(* Logix 5000 project; controller WWTP_SOLIDS_CLX vendor 1 type 14 code 54 rev 17.2; software revision 17.00; part 4 of 16 *)

ADD_ON_INSTRUCTION P_DoseFM   (* revision 0.12, ExecutePrescan, ExecuteEnableInFalse *)
// Dosing with Flowmeter
// Revision note:
// Cleaned up rate, qty code; added checks for Inp PVs being Infinite or Not A Number.
// Help:
// This Instruction monitors a flowmeter which provides flow rate (AI),
// quantity pulses (e.g., 1756-CFM/HSC), or rate and total (fieldbus),
// and provides:
// *  Optional integration (totalizing) of analog flow to a Quantity
// *  Optional differentiation of pulse count or quantity to a flow Rate
// *  Commands to Start, Stop and Clear the Quantity (total)
// *  Outputs to run and clear an external totalizer (e.g. on a fieldbus flowmeter)
// *  Commands to Start and Stop Flow for a dose
// *  Optional switching to a slow delivery (dribble) when approaching setpoint
// *  Stopping flow just before reaching setpoint using a Preact value
// *  Optional automatic adjustment of the preact value to fine tune the stop point
// *  Commands to check if the delivered quantity is within user-specified tolerances and alarm if not
// *  Program and Operator Settings for Setpoint, Preact, Dribble Quantity, High and Low Tolerances
// *  Zero failure alarm if quantity does not zero when totalizer is cleared
// *  Configurable Low Flow Cutoff to account for zero error on analog flowmeters
// *  Conversion of flow units to alternate quantity units (say, GPM to Barrels)
// *  Monitoring of input communication status
// *  Mode selection (Operator, Program or Maintenance)
// *  Simulation using configured simulated Delivery Rate and simulated Dribble Rate
VAR_INPUT
   Inp_RatePV : REAL; {visible}   // Flow Rate from Flowmeter (EU/time, see Cfg_RateTime)
   Inp_QtyPV : REAL; {visible}   // Quantity from Flowmeter (EU or Pulse Count)
   Inp_RatePVBad : BOOL;   // 1=Rate PV Input Quality = Bad (fail)
   Inp_RatePVUncertain : BOOL;   // 1=Rate PV Input Quality = Uncertain
   Inp_QtyPVBad : BOOL;   // 1=Quantity PV Input Quality = Bad (fail)
   Inp_QtyPVUncertain : BOOL;   // 1=Quantity PV Input Quality = Uncertain
   Inp_CtrldEqpFault : BOOL; {visible}   // Controlled Equipment device or I/O status 0=OK, 1=fail
   Inp_Sim : BOOL;   // 1=Simulate working flowmeter; 0=use actual flowmeter
   Inp_Reset : BOOL; {visible}   // 1=Reset all fault conditions and latched Alarms
   Cfg_HasDribble : BOOL;   // 1=Slow to Dribble before complete, 0=use complete only
   Cfg_AutoAdjPreact : BOOL;   // 1=enable automatic adjustment of preact after each delivery
   Cfg_CalcRate : BOOL := 1;   // 1=differentiate Inp_Qty to get rate, 0=use Inp_Rate
   Cfg_CalcQty : BOOL;   // 1=integrate Inp_Rate to get Quantity, 0=use Inp_Qty
   Cfg_SetTrack : BOOL := 1;   // 1=PSets track OSets in Oper, OSets track PSets in Prog, 0=no tracking
   Cfg_PCmdClear : BOOL := 1;   // 1=Clear Program Commands on receipt 0=Leave Set
   Cfg_HasOverTolAlm : BOOL;   // 1=Over Tolerance Alarm exists and will be checked
   Cfg_HasUnderTolAlm : BOOL;   // 1=Under Tolerance Alarm exists and will be checked
   Cfg_HasZeroFaultAlm : BOOL;   // 1=Zero Fault Alarm exists and will be checked
   Cfg_HasEqpFaultAlm : BOOL;   // 1=Equipment Fault Alarm exists and will be checked
   Cfg_OverTolResetReqd : BOOL;   // 1=Reset requied to clear Out of Tolerance High Alarm
   Cfg_UnderTolResetReqd : BOOL;   // 1=Reset required to clear Out of Tolerance Low Alarm
   Cfg_ZeroFaultResetReqd : BOOL;   // 1=Reset required to clear Zero Fault Alarm
   Cfg_EqpFaultResetReqd : BOOL;   // 1=Reset required to clear Equipment Fault Alarm
   Cfg_OverTolAckReqd : BOOL := 1;   // 1=Acknowledge required for Out of Tolerance High Alarm
   Cfg_UnderTolAckReqd : BOOL := 1;   // 1=Acknowledge required for Out of Tolerance Low Alarm
   Cfg_ZeroFaultAckReqd : BOOL := 1;   // 1=Acknowledge required for Zero Fault Alarm
   Cfg_EqpFaultAckReqd : BOOL := 1;   // 1=Acknowledge required for Equipment Fault Alarm
   Cfg_OverTolSeverity : SINT := 3;   // Over Tolerance Alarm Severity 1=info, 2=warn, 3=excep, 4=fault
   Cfg_UnderTolSeverity : SINT := 2;   // Under Tolerance Alarm Severity 1=info, 2=warn, 3=excep, 4=fault
   Cfg_ZeroFaultSeverity : SINT := 4;   // Zero Fault Alarm Severity 1=info, 2=warn, 3=excep, 4=fault
   Cfg_EqpFaultSeverity : SINT := 4;   // Equipment Fault Alarm Severity 1=info, 2=warn, 3=excep, 4=fault
   Cfg_MaxQty : REAL := 1.5e+38;   // Maximum allowed quantity to deliver (setpoint) (EU)
   Cfg_EUQtyMult : REAL := 1.0;   // Rate to Quantity EU Multiplier (e.g., Gal to Bbl.)
   Cfg_Rollover : REAL;   // Quantity Rollover (e.g., total counts for pulse input)
   Cfg_CountsPerEU : REAL := 1.0;   // Number of Counts in Inp_QtyPV which equal 1.0 EU
   Cfg_RateTime : REAL := 1.0;   // Time factor for rate (60 for /min, 3600 for /hr) (Sec)
   Cfg_RateFiltTC : REAL := 0.1;   // Filter Time Constant (sec) for calculated Rate
   Cfg_LoRateCutoff : REAL;   // Rate below which to report zero flow (Inp_RatePV untis)
   Cfg_BumpT : REAL;   // Bump (manual top-off) Time (Sec)
   Cfg_AutoAdjPct : REAL := 10.0;   // Percentage of delivery error to auto-adjust preact (%)
   Cfg_SimRate : REAL := 1.0;   // Rate at which to deliver when running in Simulation (EU/rate time)
   Cfg_SimDribbleRate : REAL := 0.1;   // Rate at which to dribble when running in Simulation (EU/rate time)
   Cfg_ClearPulseT : DINT := 1;   // Time to pulse Out_Clear to clear external totalizer (sec)
   PSet_SP : REAL;   // Program Setting of total quantity to deliver (EU)
   PSet_DribbleQty : REAL;   // Program Setting of quantity to dribble (EU)
   PSet_Preact : REAL;   // Program Setting of amount before total to stop flow (EU)
   PSet_TolHi : REAL;   // Program Setting of High Tolerance Limit (OK amount > SP)
   PSet_TolLo : REAL;   // Program Setting of Low Tolerance Limit (OK amount < SP)
   PSet_Owner : DINT;   // Program Owner Request ID (non-zero) or Release (zero)
   OSet_SP : REAL;   // Operator Setting of total quantity to deliver (EU)
   OSet_DribbleQty : REAL;   // Operator Setting of quantity to dribble (EU)
   OSet_Preact : REAL;   // Operator Setting of amount before total to stop flow (EU)
   OSet_TolHi : REAL;   // Operator Setting of High Tolerance Limit (OK amount > SP)
   OSet_TolLo : REAL;   // Operator Setting of Low Tolerance Limit (OK amount < SP)
   PCmd_ClearTot : BOOL;   // Program Command to Clear Totalizer Qty
   PCmd_StartTot : BOOL;   // Program Command to Start Totalizer
   PCmd_StopTot : BOOL;   // Program Command to Stop Totalizer
   PCmd_StartFlow : BOOL;   // Program Command to Start Delivery
   PCmd_StopFlow : BOOL;   // Program Command to Stop/Pause Delivery
   PCmd_CheckTol : BOOL;   // Program Command to Check Tolerances
   PCmd_Acq : BOOL;   // Program Command to Acquire ownership (Oper/OOS to Prog)
   PCmd_Rel : BOOL;   // Program Command to Release ownership (Prog to OOS)
   PCmd_Lock : BOOL;   // Program Command to Lock Mode in Prog
   PCmd_Unlock : BOOL;   // Program Command to Unlock Mode
   PCmd_Reset : BOOL;   // Program Command to Reset all Alarms requiring Reset
   PCmd_OverTolAck : BOOL;   // Program Command to Acknowledge Out of Tolerance High Alarm
   PCmd_OverTolInhibit : BOOL;   // Program Command to Inhibit Out of Tolerance High Alarm
   PCmd_OverTolUninhibit : BOOL;   // Program Command to Uninhibit Out of Tolerance High Alarm
   PCmd_UnderTolAck : BOOL;   // Program Command to Acknowledge Out of Tolerance Low Alarm
   PCmd_UnderTolInhibit : BOOL;   // Program Command to Inhibit Out of Tolerance Low Alarm
   PCmd_UnderTolUninhibit : BOOL;   // Program Command to Uninhibit Out of Tolerance Low Alarm
   PCmd_ZeroFaultAck : BOOL;   // Program Command to Acknowledge Zero Fault Alarm
   PCmd_ZeroFaultInhibit : BOOL;   // Program Command to Inhibit Zero Fault Alarm
   PCmd_ZeroFaultUninhibit : BOOL;   // Program Command to Uninhibit Zero Fault Alarm
   PCmd_EqpFaultAck : BOOL;   // Program Command to Acknowledge Equipment Fault Alarm
   PCmd_EqpFaultInhibit : BOOL;   // Program Command to Inhibit Equipment Fault Alarm
   PCmd_EqpFaultUninhibit : BOOL;   // Program Command to Uninhibit Equipment Fault Alarm
   OCmd_ClearTot : BOOL;   // Operator Command to Clear Totalizer Qty
   OCmd_StartTot : BOOL;   // Operator Command to Start Totalizer
   OCmd_StopTot : BOOL;   // Operator Command to Stop Totalizer
   OCmd_StartFlow : BOOL;   // Operator command to Start Deliver
   OCmd_StopFlow : BOOL;   // Operator Command to Stop/Pause Delivery
   OCmd_CheckTol : BOOL;   // Operator Command to Check Tolerances
   OCmd_Bump : BOOL;   // Operator Command to Bump Delivery for Under Tolerance
   OCmd_Reset : BOOL;   // Operator Command to Reset all Alarms requiring Reset
END_VAR
VAR_OUTPUT
   Out_RunFlow : BOOL; {visible}   // 1=Deliver at Full (fast) Flow
   Out_DribbleFlow : BOOL; {visible}   // 1=Deliver at Dribble (slow) Flow
   Out_StopFlow : BOOL; {visible}   // 1=Stop Delivery Equipment
   Out_RunTot : BOOL;   // 1=Run external totalizer (e.g. onboard flowmeter)
   Out_ClearTot : BOOL;   // 1=Reset external totalizer (e.g. onboard flowmeter)
   Val_Qty : REAL; {visible}   // Quantity actually delivered (totalizer output) (EU)
   Val_Rate : REAL; {visible}   // Current Delivery Rate (EU/time) (see Cfg_RateTime)
   Val_Remain : REAL; {visible}   // Amount yet to deliver to reach Setpoint (EU)
   Val_PctComplete : REAL; {visible}   // Percent Complete (for Progress Bar on HMI) 0.0 to 100.0%
   Val_SP : REAL; {visible}   // Amount to be delivered (Setpoint) (EU)
   Val_DribbleQty : REAL; {visible}   // Amount to be delivered at slow rate (EU)
   Val_Preact : REAL; {visible}   // Amount before SP at which flow will be stopped (EU)
   Val_TolHi : REAL; {visible}   // Allowed Amount > SP (EU)
   Val_TolLo : REAL; {visible}   // Allowed Amount < SP (EU)
   Val_Owner : DINT;   // Current Object Owner ID (0=not owned)
   Val_Notify : SINT;   // Current Alarm Level and Acknowledgement (enumeration)
   Sts_Cleared : BOOL; {visible}   // 1=Totalizer Clear completed
   Sts_TotRunning : BOOL; {visible}   // 1=Totalizer Running, 0=Totalizer Stopped
   Sts_FlowRunning : BOOL; {visible}   // 1=Flow is Running (Out_Run is ON)
   Sts_FlowDribble : BOOL; {visible}   // 1=Flow is slowed to Dribble (Out_Dribble is ON)
   Sts_FlowStopped : BOOL; {visible}   // 1=Flow is Stopped (Out_Stop is ON)
   Sts_Bumping : BOOL;   // 1=Bump flow (timed) is active
   Sts_LoRateCutoff : BOOL;   // 1=Rate PV below low rate cutoff, flow assumed to be zero
   Sts_Complete : BOOL; {visible}   // 1=Total Delivered > (SP - Preact)
   Sts_InTol : BOOL;   // 1=Total Delivered is Within Tolerances
   Sts_Available : BOOL;   // 1=Dosing available for control by automation (Prog)
   Sts_QtyBad : BOOL;   // 1=Quantity Value is Bad (PV Fail)
   Sts_QtyUncertain : BOOL;   // 1=Quantity Value is Uncertain
   Sts_RateBad : BOOL;   // 1=Rate Value is Bad (PV Fail)
   Sts_RateUncertain : BOOL;   // 1=Rate Value is Uncertain
   Sts_Err : BOOL; {visible}   // 1=Error: Bad Configuration, see detail Err bits for reason
   Err_EU : BOOL;   // 1=Error: Cfg_CountsPerEU, Cfg_EUQtyMult or Cfg_Rollowver invalid
   Err_Rate : BOOL;   // 1=Error: Cfg_RateFiltTC or Cfg_RateTime invalid
   Err_Cutoff : BOOL;   // 1=Error: Cfg_LoRateCutoff invalid
   Err_Limit : BOOL;   // 1=Error: Cfg_MaxQty invalid
   Err_Sim : BOOL;   // 1=Error: Cfg_SimDribbleRate or Cfg_SimRate invalid
   Err_Timer : BOOL;   // 1=Error: Cfg_BumpT or Cfg_ClearPulseT (use 0.0 to 2147483.647)
   Err_Alarm : BOOL;   // 1=Error: Alarm Severity Cfg Invalid
   Sts_Maint : BOOL; {visible}   // 1=Mode is Maintenance (supersedes Prog, Oper)
   Sts_Prog : BOOL; {visible}   // 1=Mode is Program (auto)
   Sts_Oper : BOOL := 1; {visible}   // 1=Mode is Operator (manual)
   Sts_ProgOperLock : BOOL;   // 1=Program or Operator has requested Mode Lock
   Sts_OverTol : BOOL;   // 1=Delivery Out of Tolerance High
   Alm_OverTol : BOOL;   // 1=Delivery Out of Tolerance High Alarm
   Ack_OverTol : BOOL;   // 1=Out of Tolerance High Alarm has been acknowledged
   Sts_OverTolDisabled : BOOL;   // 1=Out of Tolerance High Alarm has been disabled (will not be sent)
   Sts_OverTolInhibited : BOOL;   // 1=Out of Tolerance High Alarm has been inhibited by logic
   Sts_OverTolSuppressed : BOOL;   // 1=Out of Tolerance High Alarm has been suppressed (logged only)
   Sts_UnderTol : BOOL;   // 1=Delivery Out of Tolerance Low
   Alm_UnderTol : BOOL;   // 1=Delivery Out of Tolerance Low Alarm
   Ack_UnderTol : BOOL;   // 1=Out of Tolerance Low Alarm has been acknowledged
   Sts_UnderTolDisabled : BOOL;   // 1=Out of Tolerance Low Alarm has been disabled (will not be sent)
   Sts_UnderTolInhibited : BOOL;   // 1=Out of Tolerance Low Alarm has been inhibited by logic
   Sts_UnderTolSuppressed : BOOL;   // 1=Out of Tolerance Low Alarm has been suppressed (logged only)
   Sts_ZeroFault : BOOL;   // 1=Total did not clear or unexpected flow
   Alm_ZeroFault : BOOL;   // 1=Warning: Total did not clear or still flowing
   Ack_ZeroFault : BOOL;   // 1=Zero Fault Alarm has been acknowledged
   Sts_ZeroFaultDisabled : BOOL;   // 1=Zero Fault Alarm is Disabled (not saved or sent)
   Sts_ZeroFaultInhibited : BOOL;   // 1=Zero Fault Alarm has been inhibited by logic
   Sts_ZeroFaultSuppressed : BOOL;   // 1=Zero Fault Alarm has been suppressed (logged only)
   Sts_EqpFault : BOOL;   // 1=Equipment Fault Detected
   Alm_EqpFault : BOOL;   // 1=Equipment Fault Alarm
   Ack_EqpFault : BOOL;   // 1=Equipment Fault Alarm has been acknowledged
   Sts_EqpFaultDisabled : BOOL;   // 1=Equipment Fault Alarm is Disabled (not saved or sent)
   Sts_EqpFaultInhibited : BOOL;   // 1=Equipment Fault Alarm has been inhibited by logic
   Sts_EqpFaultSuppressed : BOOL;   // 1=Equipment Fault Alarm has been suppressed (logged only)
   Rdy_ClearTot : BOOL;   // 1=Ready for OCmd_ClearTot (enables button)
   Rdy_StartTot : BOOL;   // 1=Ready for OCmd_StartTot (enables button)
   Rdy_StopTot : BOOL;   // 1=Ready for OCmd_StopTot (enables button)
   Rdy_StartFlow : BOOL;   // 1=Ready for OCmd_StartFlow (enables button)
   Rdy_StopFlow : BOOL;   // 1=Ready for OCmd_StopFlow (enables button)
   Rdy_CheckTol : BOOL;   // 1-Ready for OCmd_CheckTol (enables button)
   Rdy_Bump : BOOL;   // 1=Ready for OCmd_Bump (enables button)
   Rdy_Reset : BOOL;   // 1=Ready for OCmd_Reset (enables button)
END_VAR
VAR
   Cfg_RateEU : STRING_8 := 'kg/sec';   // Engineering Units for Rate (flow) for display on HMI
   Cfg_Tag : STRING_20 := 'P_DoseFM';   // Tagname for display on HMI
   Cfg_Label : STRING_20 := 'Flowmeter Dosing';   // Label for graphic symbol displayed on HMI
   Cfg_QtyEU : STRING_8 := 'kg';   // Engineering Units for Quantity for display on HMI
   Cfg_Desc : STRING_40 := 'Dosing with Flowmeter';   // Description for display on HMI
   Wrk_Notify : DINT;   // Buffer for building Val_Notify
   Mode : P_Mode := (Cfg_PCmdClear := 1, Cfg_OvrdOverLock := 1, Sts_Oper := 1, Rdy_Rel := 1, Rdy_AcqLock := 1);   // Analog Input Mode Selection
   Wrk_ClearTot : BOOL;   // Request to Clear Total received
   ZeroFault : P_Alarm := (Inp := 1, Cfg_AckReqd := 1, Cfg_Severity := 3, Ack := 1, Rdy_Disable := 1);   // Rate Not Zero when Expected Alarm
   UnderTol : P_Alarm := (Inp := 1, Cfg_AckReqd := 1, Cfg_Severity := 3, Ack := 1, Rdy_Disable := 1);   // Final Quantity Below Low Tolerance Alarm
   OverTol : P_Alarm := (Inp := 1, Cfg_AckReqd := 1, Cfg_Severity := 3, Ack := 1, Rdy_Disable := 1);   // Final Quantity Above High Tolerance Alarm
   EqpFault : P_Alarm := (Inp := 1, Cfg_AckReqd := 1, Cfg_Severity := 3, Ack := 1, Rdy_Disable := 1);   // Equipment (Sensor, Controlled Equip.) Fault Alarm
   Wrk_RunFlow : BOOL;   // 1=Flow (full)( should be running
   Wrk_RunTot : BOOL;   // 1=Totalizaer should be ruuuning
   Wrk_BumpFlow : BOOL;   // Operator requested bump flow to make up Under Tolerance
   Wrk_BumpT : TIMER;   // Bump Timer for shot of flow to make up Under Tolerance
   Wrk_ClearPulseT : TIMER := (PRE := 1000);   // Time to pulse Out_Clear to clear external timer
   Wrk_ScanTime : REAL;   // Time since previous scan (sec)
   Wrk_PrevQty : REAL;   // Previous scan's Inp_QtyPV value
   Wrk_Rate : REAL;   // Instantaneous Rate based on change in Inp_Qty
   Wrk_AmtToAdd : REAL;   // Amount to add to Quantity this scan based on Rate
   Wrk_LoOrderTot : REAL;   // Fractional Amount of Totalizer (low-order of cascaded registers)
   Wrk_HiOrderTot : DINT;   // Integer Amount of Totalizer (high-order of cascaded registers)
   Wrk_PctComplete : REAL;   // Percent Complete calculation intermediate
   Wrk_BumpNoAdj : BOOL;   // Do NOT auto-adjust Preact if flow was Bumped since Clearing Totalizer
   Wrk_ScanT : TIMER := (PRE := 2147483647);   // Scan Timer (milliseconds, always runs)
   Wrk_Alpha : REAL;   // Filter multiplier = (1 / (1+TC/dT) )
   Wrk_FiltRate : REAL;   // Working register for calculating filtered delivery rate
   Wrk_RateInfNaN : BOOL;   // Rate PV is Infinite or NaN
   Wrk_RateInpDINT : DINT;   // Inp_RatePV check for Infinite or Not A Number
   Wrk_QtyInfNaN : BOOL;   // Quantity PV is Infinite or NaN
   Wrk_QtyInpDINT : DINT;   // Inp_QtyPV check for Infinite or Not A Number
   Wrk_ValidONS : BOOL;   // Rate PV goes from Infinite or Not a Number to VALID
END_VAR

ROUTINE EnableInFalse   (* ladder *)
// Clear any "lurking" Commands and all Readies, set NO MODE
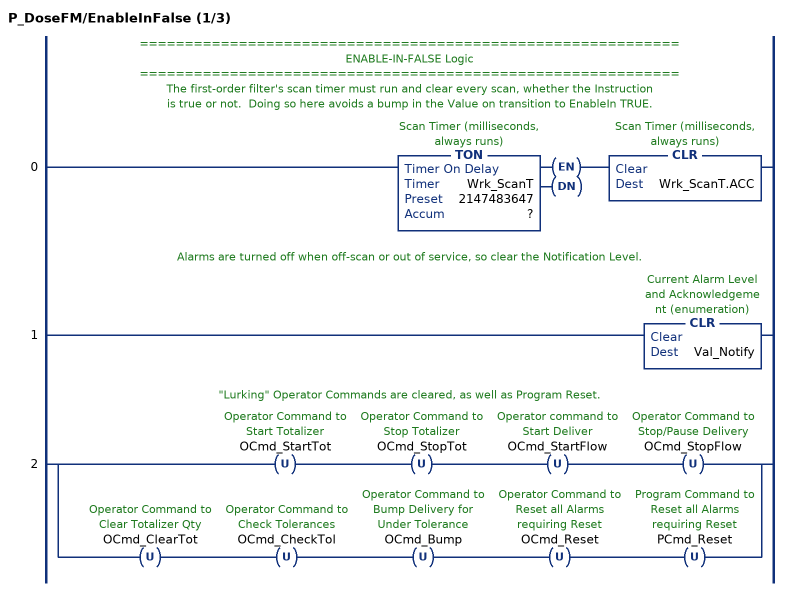
   // ============================================================
   // ENABLE-IN-FALSE Logic
   // ============================================================
   // The first-order filter's scan timer must run and clear every scan, whether the Instruction
   // is true or not.  Doing so here avoids a bump in the Value on transition to EnableIn TRUE.
   0: TON(Wrk_ScanT,?,?)CLR(Wrk_ScanT.ACC);
   // Alarms are turned off when off-scan or out of service, so clear the Notification Level.
   1: CLR(Val_Notify);
   // "Lurking" Operator Commands are cleared, as well as Program Reset.
   2: [OTU(OCmd_StartTot) OTU(OCmd_StopTot) OTU(OCmd_StartFlow) OTU(OCmd_StopFlow) ,OTU(OCmd_ClearTot) OTU(OCmd_CheckTol) OTU(OCmd_Bump) OTU(OCmd_Reset) OTU(PCmd_Reset) ];
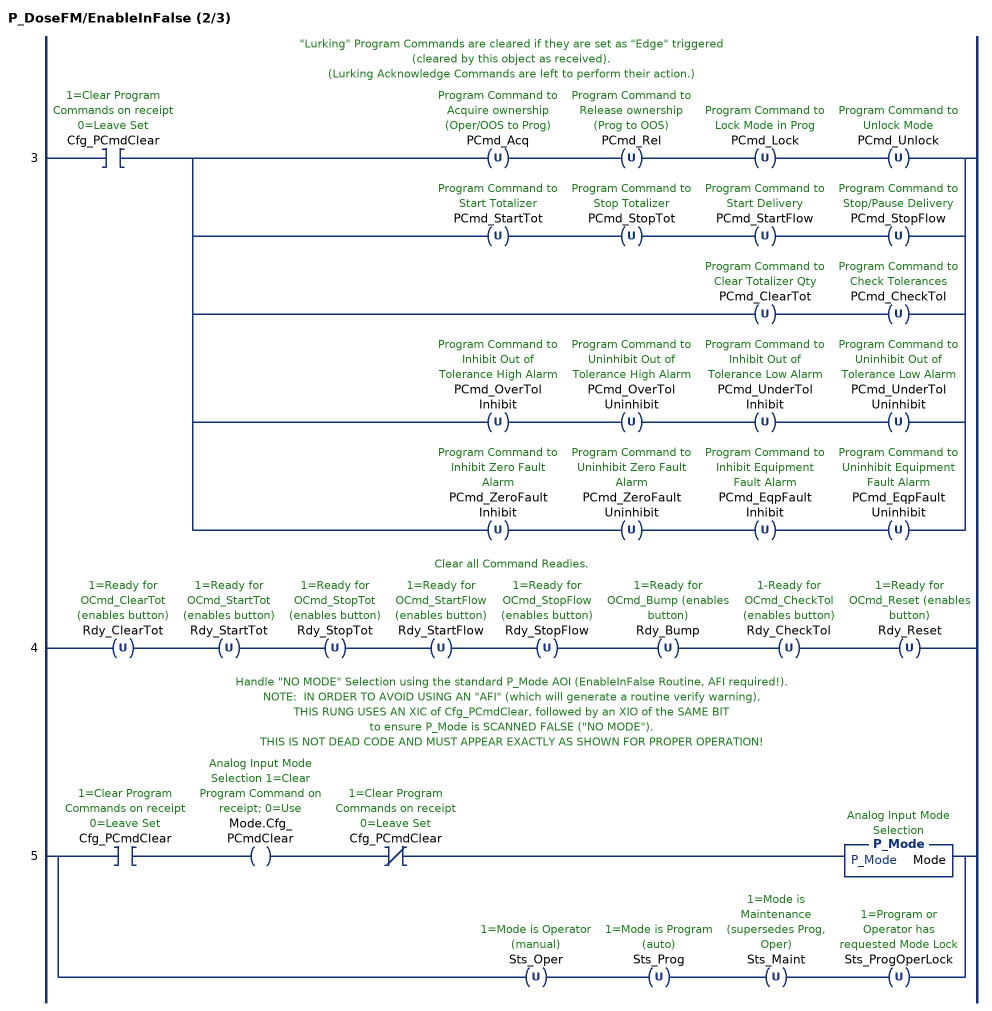
   // "Lurking" Program Commands are cleared if they are set as "Edge" triggered
   // (cleared by this object as received).
   // (Lurking Acknowledge Commands are left to perform their action.)
   3: XIC(Cfg_PCmdClear)[OTU(PCmd_Acq) OTU(PCmd_Rel) OTU(PCmd_Lock) OTU(PCmd_Unlock) ,OTU(PCmd_StartTot) OTU(PCmd_StopTot) OTU(PCmd_StartFlow) OTU(PCmd_StopFlow) ,OTU(PCmd_ClearTot) OTU(PCmd_CheckTol) ,OTU(PCmd_OverTolInhibit) OTU(PCmd_OverTolUninhibit) OTU(PCmd_UnderTolInhibit) OTU(PCmd_UnderTolUninhibit) ,OTU(PCmd_ZeroFaultInhibit) OTU(PCmd_ZeroFaultUninhibit) OTU(PCmd_EqpFaultInhibit) OTU(PCmd_EqpFaultUninhibit) ];
   // Clear all Command Readies.
   4: OTU(Rdy_ClearTot)OTU(Rdy_StartTot)OTU(Rdy_StopTot)OTU(Rdy_StartFlow)OTU(Rdy_StopFlow)OTU(Rdy_Bump)OTU(Rdy_CheckTol)OTU(Rdy_Reset);
   // Handle "NO MODE" Selection using the standard P_Mode AOI (EnableInFalse Routine, AFI required!).
   // NOTE:  IN ORDER TO AVOID USING AN "AFI" (which will generate a routine verify warning),
   // THIS RUNG USES AN XIC of Cfg_PCmdClear, followed by an XIO of the SAME BIT
   // to ensure P_Mode is SCANNED FALSE ("NO MODE").
   // THIS IS NOT DEAD CODE AND MUST APPEAR EXACTLY AS SHOWN FOR PROPER OPERATION!
   5: [XIC(Cfg_PCmdClear) OTE(Mode.Cfg_PCmdClear) XIO(Cfg_PCmdClear) P_Mode(Mode) ,OTU(Sts_Oper) OTU(Sts_Prog) OTU(Sts_Maint) OTU(Sts_ProgOperLock) ];
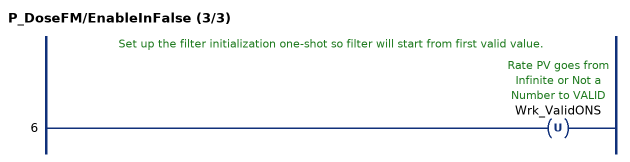
   // Set up the filter initialization one-shot so filter will start from first valid value.
   6: OTU(Wrk_ValidONS);
END_ROUTINE

ROUTINE Logic   (* ladder *)
// Normal Scan: control / monitor Dosing with Flowmeter
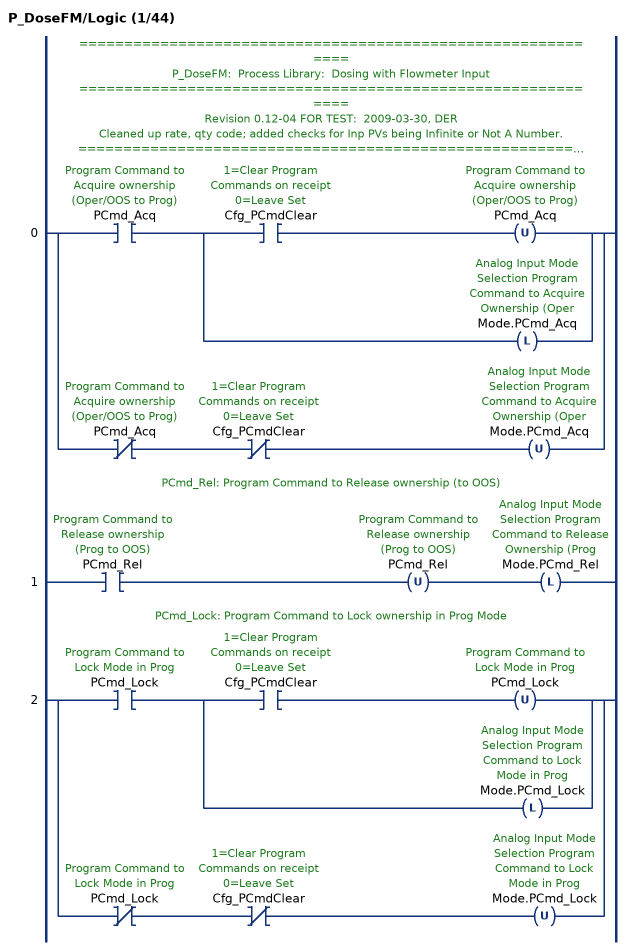
   // ============================================================
   // P_DoseFM:  Process Library:  Dosing with Flowmeter Input
   // ============================================================
   // Revision 0.12-04 FOR TEST:  2009-03-30, DER
   // Cleaned up rate, qty code; added checks for Inp PVs being Infinite or Not A Number.
   // ============================================================
   // This Instruction monitors a flowmeter which provides flow rate (AI),
   // quantity pulses (e.g., 1756-CFM / -HSC), or rate and total (fieldbus),
   // and provides:
   // *  Optional integration (totalizing) of analog flow to a Quantity
   // *  Optional differentiation of pulse count or quantity to a flow Rate
   // *  Commands to Start, Stop and Clear the Quantity (total)
   // *  Outputs to run and clear an external totalizer (say, on fieldbus flowmeter)
   // *  Commands to Start and Stop Flow for a dosing
   // *  Optional switching to a slow delivery (dribble) when approaching setpoint
   // *  Stopping flow just before reaching setpoint using a Preact value
   // *  Optional automatic adjustment of the preact value to fine tune the stop point
   // *  Commands to check if the delivered quantity is within user-specified tolerances and alarm if not
   // *  Program and Operator Settings for Setpoint, Preact, Dribble Quantity, High and Low Tolerances
   // *  Equipment Failure Alarm on sensor failure (stops totalizer, stops flow) or controlled equipment failure (stops flow)
   // *  Zero failure alarm if quantity does not zero when totalizer is cleared
   // *  Configurable Low Flow Cutoff to account for zero error on analog flowmeters
   // *  Conversion of flow units to alternate quantity units (e.g., GPM to Barrels)
   // *  Mode selection (Operator, Program or Maintenance)
   // *  Simulation using a provided simulated Rate and simulated Dribble Rate
   // ============================================================
   // POWERUP / INVALID STATE HANDLING
   // ============================================================
   // Mode states are retained through a power cycle.
   // No special powerup code is required for this object.
   // ============================================================
   // MODE PROCESSING
   // ============================================================
   // These rungs handle received Mode Inputs and Commands:
   // NOTE:  Operator Commands for Mode, Alarm are sent directly to the contained P_Mode and P_Alarm AOIs.
   // PCmd_Acq: Program Command to Acquire ownership
   0: [XIC(PCmd_Acq) [XIC(Cfg_PCmdClear) OTU(PCmd_Acq) ,OTL(Mode.PCmd_Acq) ] ,XIO(PCmd_Acq) XIO(Cfg_PCmdClear) OTU(Mode.PCmd_Acq) ];
   // PCmd_Rel: Program Command to Release ownership (to OOS)
   1: XIC(PCmd_Rel)OTU(PCmd_Rel)OTL(Mode.PCmd_Rel);
   // PCmd_Lock: Program Command to Lock ownership in Prog Mode
   2: [XIC(PCmd_Lock) [XIC(Cfg_PCmdClear) OTU(PCmd_Lock) ,OTL(Mode.PCmd_Lock) ] ,XIO(PCmd_Lock) XIO(Cfg_PCmdClear) OTU(Mode.PCmd_Lock) ];
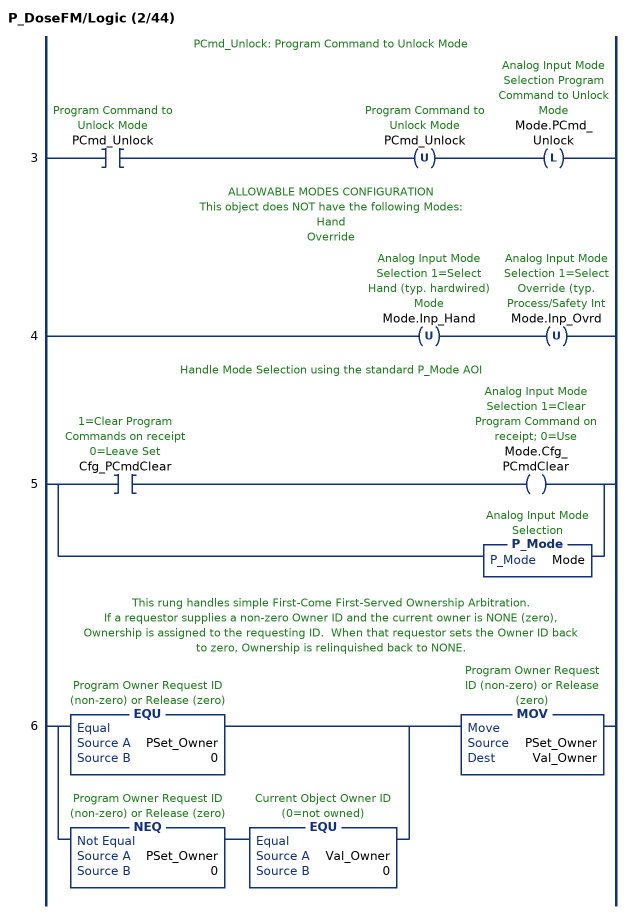
   // PCmd_Unlock: Program Command to Unlock Mode
   3: XIC(PCmd_Unlock)OTU(PCmd_Unlock)OTL(Mode.PCmd_Unlock);
   // ALLOWABLE MODES CONFIGURATION
   // This object does NOT have the following Modes:
   // Hand
   // Override
   4: OTU(Mode.Inp_Hand)OTU(Mode.Inp_Ovrd);
   // Handle Mode Selection using the standard P_Mode AOI
   5: [XIC(Cfg_PCmdClear) OTE(Mode.Cfg_PCmdClear) ,P_Mode(Mode) ];
   // This rung handles simple First-Come First-Served Ownership Arbitration.
   // If a requestor supplies a non-zero Owner ID and the current owner is NONE (zero),
   // Ownership is assigned to the requesting ID.  When that requestor sets the Owner ID back
   // to zero, Ownership is relinquished back to NONE.
   6: [EQU(PSet_Owner,0) ,NEQ(PSet_Owner,0) EQU(Val_Owner,0) ]MOV(PSet_Owner,Val_Owner);
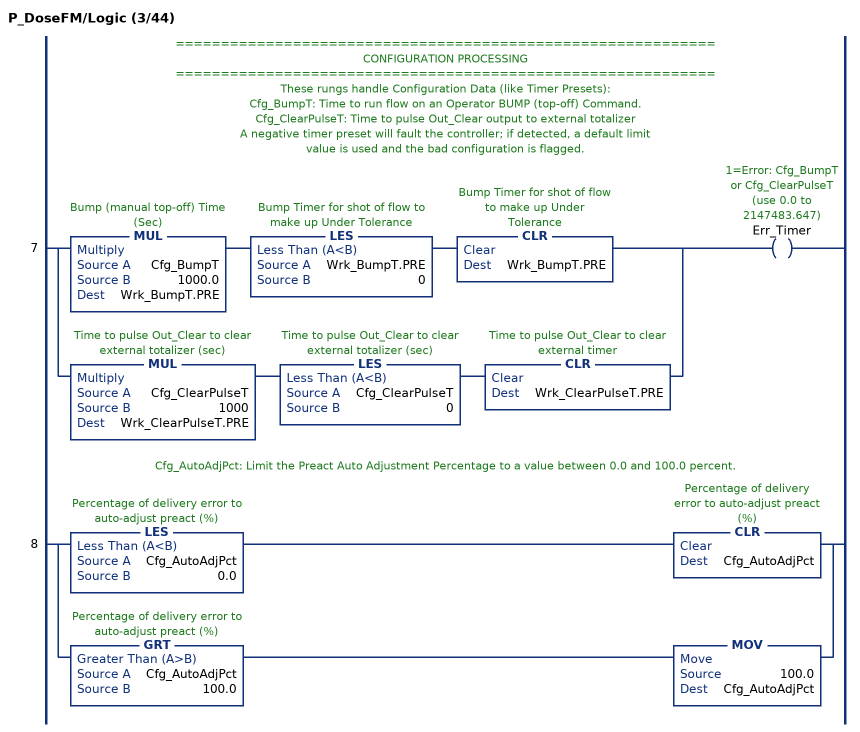
   // ============================================================
   // CONFIGURATION PROCESSING
   // ============================================================
   // These rungs handle Configuration Data (like Timer Presets):
   // Cfg_BumpT: Time to run flow on an Operator BUMP (top-off) Command.
   // Cfg_ClearPulseT: Time to pulse Out_Clear output to external totalizer
   // A negative timer preset will fault the controller; if detected, a default limit
   // value is used and the bad configuration is flagged.
   7: [MUL(Cfg_BumpT,1000.0,Wrk_BumpT.PRE) LES(Wrk_BumpT.PRE,0) CLR(Wrk_BumpT.PRE) ,MUL(Cfg_ClearPulseT,1000,Wrk_ClearPulseT.PRE) LES(Cfg_ClearPulseT,0) CLR(Wrk_ClearPulseT.PRE) ]OTE(Err_Timer);
   // Cfg_AutoAdjPct: Limit the Preact Auto Adjustment Percentage to a value between 0.0 and 100.0 percent.
   8: [LES(Cfg_AutoAdjPct,0.0) CLR(Cfg_AutoAdjPct) ,GRT(Cfg_AutoAdjPct,100.0) MOV(100.0,Cfg_AutoAdjPct) ];
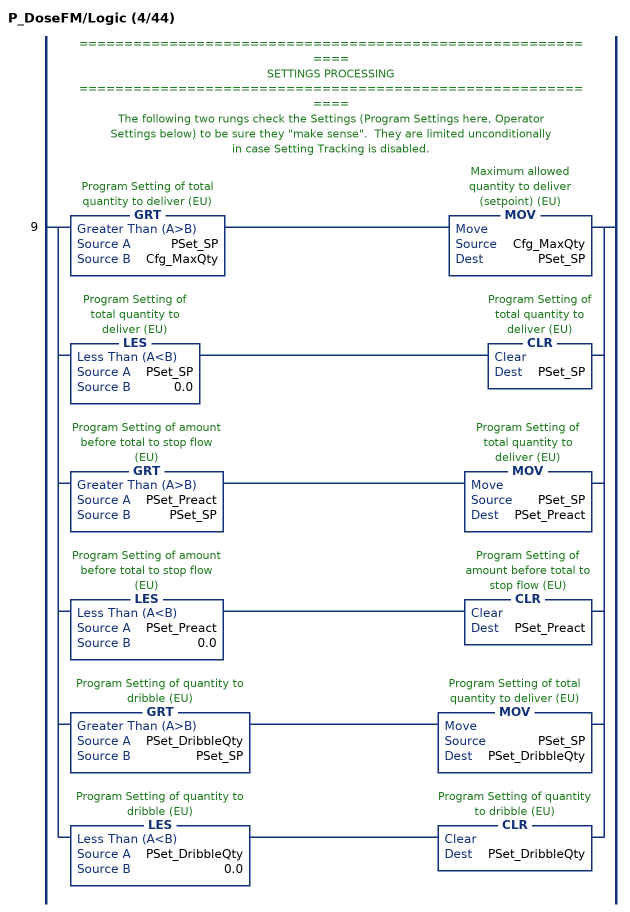
   // ============================================================
   // SETTINGS PROCESSING
   // ============================================================
   // The following two rungs check the Settings (Program Settings here, Operator
   // Settings below) to be sure they "make sense".  They are limited unconditionally
   // in case Setting Tracking is disabled.
   9: [GRT(PSet_SP,Cfg_MaxQty) MOV(Cfg_MaxQty,PSet_SP) ,LES(PSet_SP,0.0) CLR(PSet_SP) ,GRT(PSet_Preact,PSet_SP) MOV(PSet_SP,PSet_Preact) ,LES(PSet_Preact,0.0) CLR(PSet_Preact) ,GRT(PSet_DribbleQty,PSet_SP) MOV(PSet_SP,PSet_DribbleQty) ,LES(PSet_DribbleQty,0.0) CLR(PSet_DribbleQty) ];
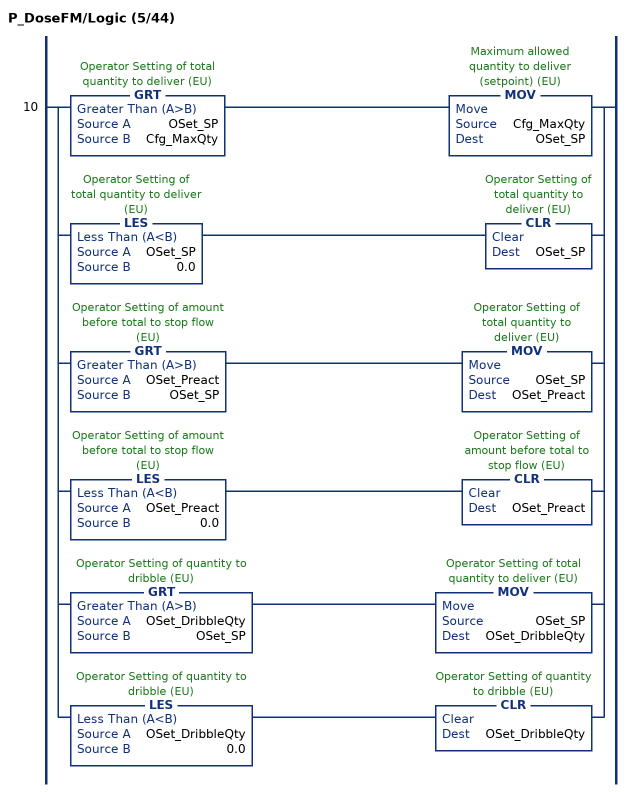
   10: [GRT(OSet_SP,Cfg_MaxQty) MOV(Cfg_MaxQty,OSet_SP) ,LES(OSet_SP,0.0) CLR(OSet_SP) ,GRT(OSet_Preact,OSet_SP) MOV(OSet_SP,OSet_Preact) ,LES(OSet_Preact,0.0) CLR(OSet_Preact) ,GRT(OSet_DribbleQty,OSet_SP) MOV(OSet_SP,OSet_DribbleQty) ,LES(OSet_DribbleQty,0.0) CLR(OSet_DribbleQty) ];
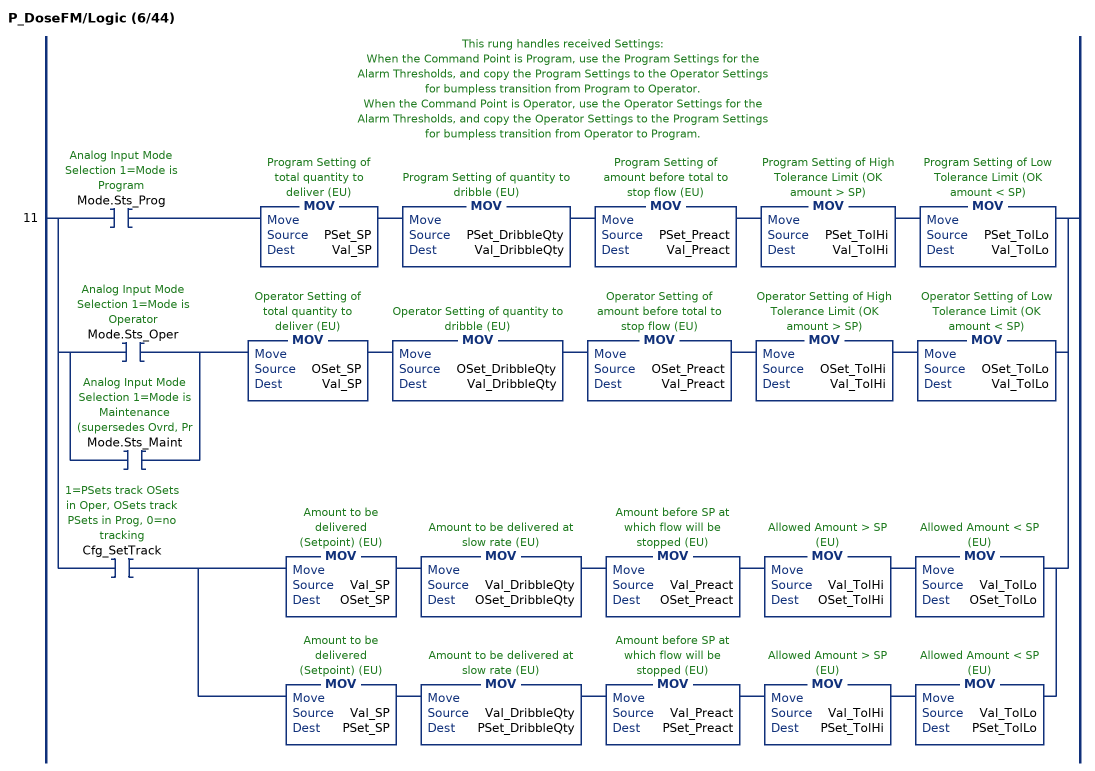
   // This rung handles received Settings:
   // When the Command Point is Program, use the Program Settings for the
   // Alarm Thresholds, and copy the Program Settings to the Operator Settings
   // for bumpless transition from Program to Operator.
   // When the Command Point is Operator, use the Operator Settings for the
   // Alarm Thresholds, and copy the Operator Settings to the Program Settings
   // for bumpless transition from Operator to Program.
   11: [XIC(Mode.Sts_Prog) MOV(PSet_SP,Val_SP) MOV(PSet_DribbleQty,Val_DribbleQty) MOV(PSet_Preact,Val_Preact) MOV(PSet_TolHi,Val_TolHi) MOV(PSet_TolLo,Val_TolLo) ,[XIC(Mode.Sts_Oper) ,XIC(Mode.Sts_Maint) ] MOV(OSet_SP,Val_SP) MOV(OSet_DribbleQty,Val_DribbleQty) MOV(OSet_Preact,Val_Preact) MOV(OSet_TolHi,Val_TolHi) MOV(OSet_TolLo,Val_TolLo) ,XIC(Cfg_SetTrack) [MOV(Val_SP,OSet_SP) MOV(Val_DribbleQty,OSet_DribbleQty) MOV(Val_Preact,OSet_Preact) MOV(Val_TolHi,OSet_TolHi) MOV(Val_TolLo,OSet_TolLo) ,MOV(Val_SP,PSet_SP) MOV(Val_DribbleQty,PSet_DribbleQty) MOV(Val_Preact,PSet_Preact) MOV(Val_TolHi,PSet_TolHi) MOV(Val_TolLo,PSet_TolLo) ] ];
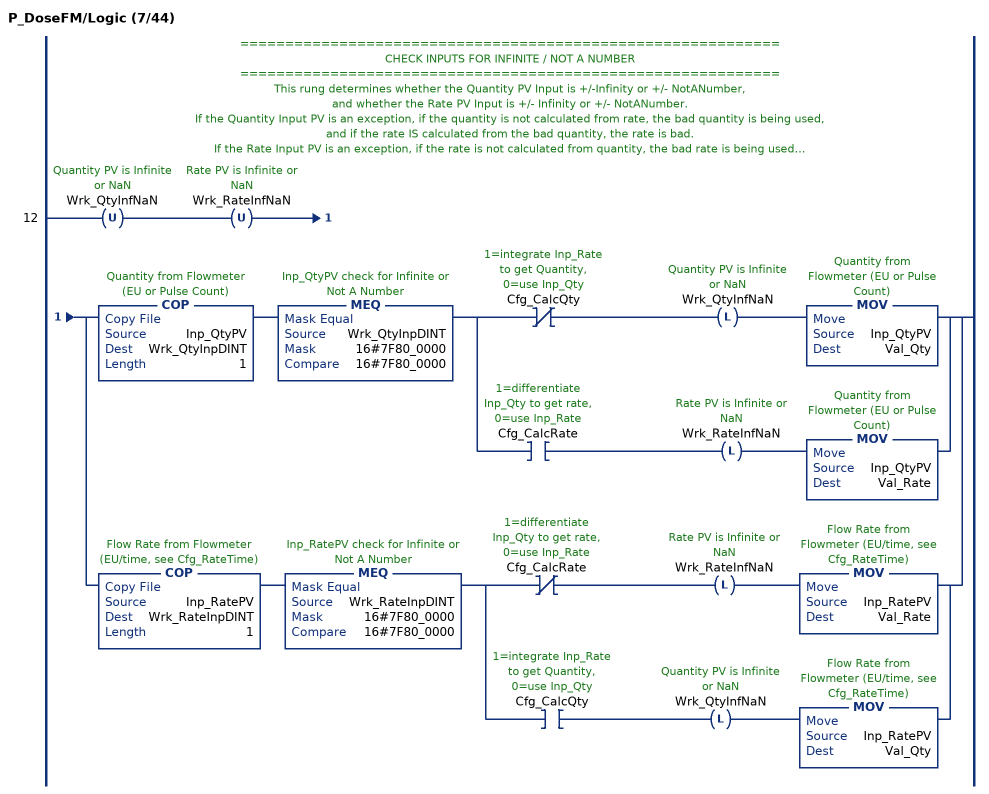
   // ============================================================
   // CHECK INPUTS FOR INFINITE / NOT A NUMBER
   // ============================================================
   // This rung determines whether the Quantity PV Input is +/-Infinity or +/- NotANumber,
   // and whether the Rate PV Input is +/- Infinity or +/- NotANumber.
   // If the Quantity Input PV is an exception, if the quantity is not calculated from rate, the bad quantity is being used,
   // and if the rate IS calculated from the bad quantity, the rate is bad.
   // If the Rate Input PV is an exception, if the rate is not calculated from quantity, the bad rate is being used,
   // and if the quantity IS calculated from the bad rate, the quantity is bad.
   12: OTU(Wrk_QtyInfNaN)OTU(Wrk_RateInfNaN)[COP(Inp_QtyPV,Wrk_QtyInpDINT,1) MEQ(Wrk_QtyInpDINT,16#7F80_0000,16#7F80_0000) [XIO(Cfg_CalcQty) OTL(Wrk_QtyInfNaN) MOV(Inp_QtyPV,Val_Qty) ,XIC(Cfg_CalcRate) OTL(Wrk_RateInfNaN) MOV(Inp_QtyPV,Val_Rate) ] ,COP(Inp_RatePV,Wrk_RateInpDINT,1) MEQ(Wrk_RateInpDINT,16#7F80_0000,16#7F80_0000) [XIO(Cfg_CalcRate) OTL(Wrk_RateInfNaN) MOV(Inp_RatePV,Val_Rate) ,XIC(Cfg_CalcQty) OTL(Wrk_QtyInfNaN) MOV(Inp_RatePV,Val_Qty) ] ];
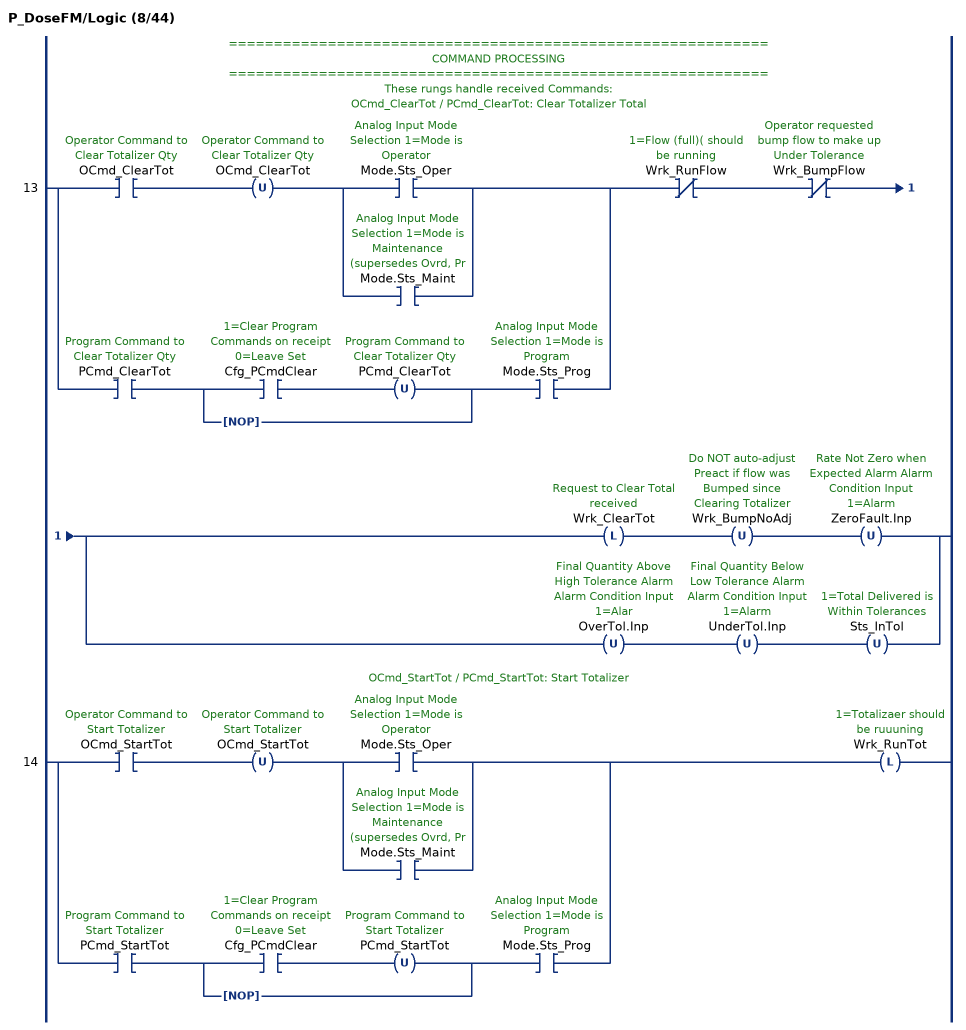
   // ============================================================
   // COMMAND PROCESSING
   // ============================================================
   // These rungs handle received Commands:
   // OCmd_ClearTot / PCmd_ClearTot: Clear Totalizer Total
   13: [XIC(OCmd_ClearTot) OTU(OCmd_ClearTot) [XIC(Mode.Sts_Oper) ,XIC(Mode.Sts_Maint) ] ,XIC(PCmd_ClearTot) [XIC(Cfg_PCmdClear) OTU(PCmd_ClearTot) ,NOP() ] XIC(Mode.Sts_Prog) ]XIO(Wrk_RunFlow)XIO(Wrk_BumpFlow)[OTL(Wrk_ClearTot) OTU(Wrk_BumpNoAdj) OTU(ZeroFault.Inp) ,OTU(OverTol.Inp) OTU(UnderTol.Inp) OTU(Sts_InTol) ];
   // OCmd_StartTot / PCmd_StartTot: Start Totalizer
   14: [XIC(OCmd_StartTot) OTU(OCmd_StartTot) [XIC(Mode.Sts_Oper) ,XIC(Mode.Sts_Maint) ] ,XIC(PCmd_StartTot) [XIC(Cfg_PCmdClear) OTU(PCmd_StartTot) ,NOP() ] XIC(Mode.Sts_Prog) ]OTL(Wrk_RunTot);
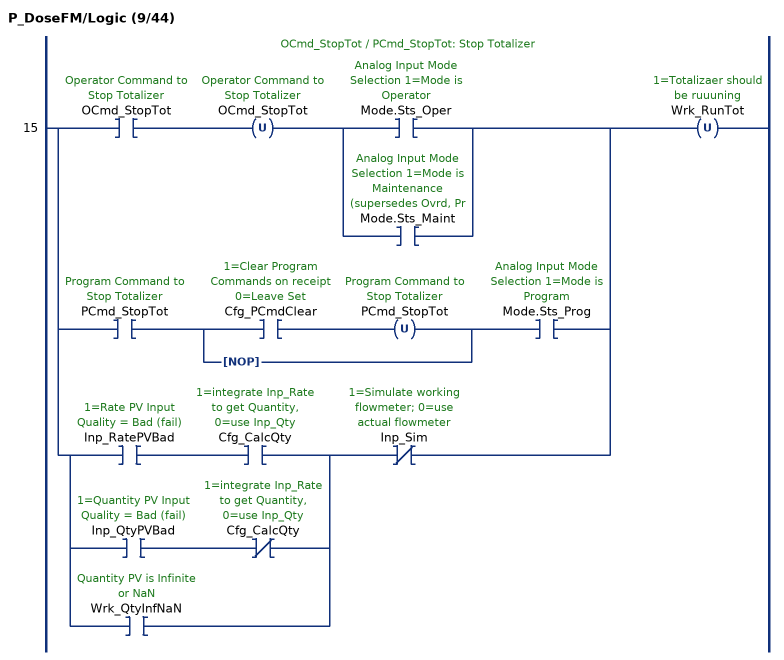
   // OCmd_StopTot / PCmd_StopTot: Stop Totalizer
   15: [XIC(OCmd_StopTot) OTU(OCmd_StopTot) [XIC(Mode.Sts_Oper) ,XIC(Mode.Sts_Maint) ] ,XIC(PCmd_StopTot) [XIC(Cfg_PCmdClear) OTU(PCmd_StopTot) ,NOP() ] XIC(Mode.Sts_Prog) ,[XIC(Inp_RatePVBad) XIC(Cfg_CalcQty) ,XIC(Inp_QtyPVBad) XIO(Cfg_CalcQty) ,XIC(Wrk_QtyInfNaN) ] XIO(Inp_Sim) ]OTU(Wrk_RunTot);
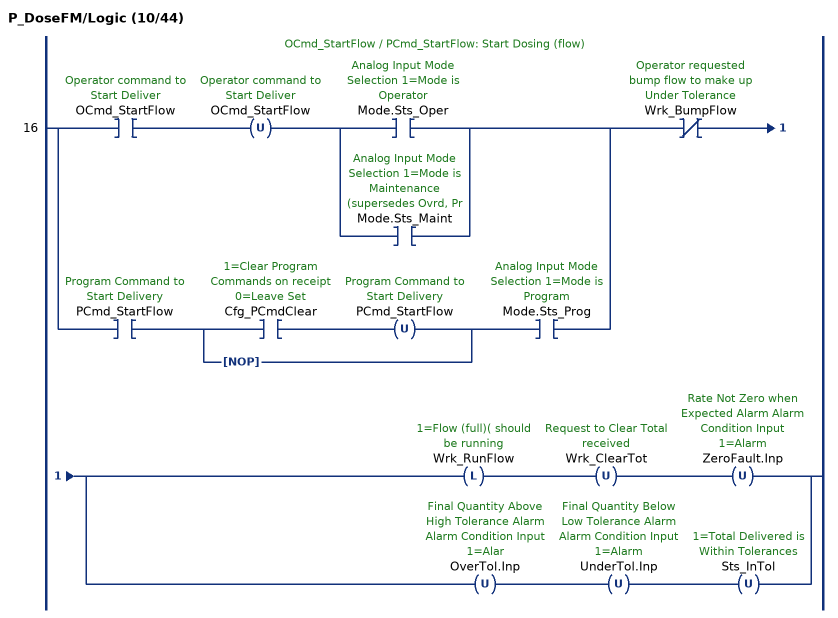
   // OCmd_StartFlow / PCmd_StartFlow: Start Dosing (flow)
   16: [XIC(OCmd_StartFlow) OTU(OCmd_StartFlow) [XIC(Mode.Sts_Oper) ,XIC(Mode.Sts_Maint) ] ,XIC(PCmd_StartFlow) [XIC(Cfg_PCmdClear) OTU(PCmd_StartFlow) ,NOP() ] XIC(Mode.Sts_Prog) ]XIO(Wrk_BumpFlow)[OTL(Wrk_RunFlow) OTU(Wrk_ClearTot) OTU(ZeroFault.Inp) ,OTU(OverTol.Inp) OTU(UnderTol.Inp) OTU(Sts_InTol) ];
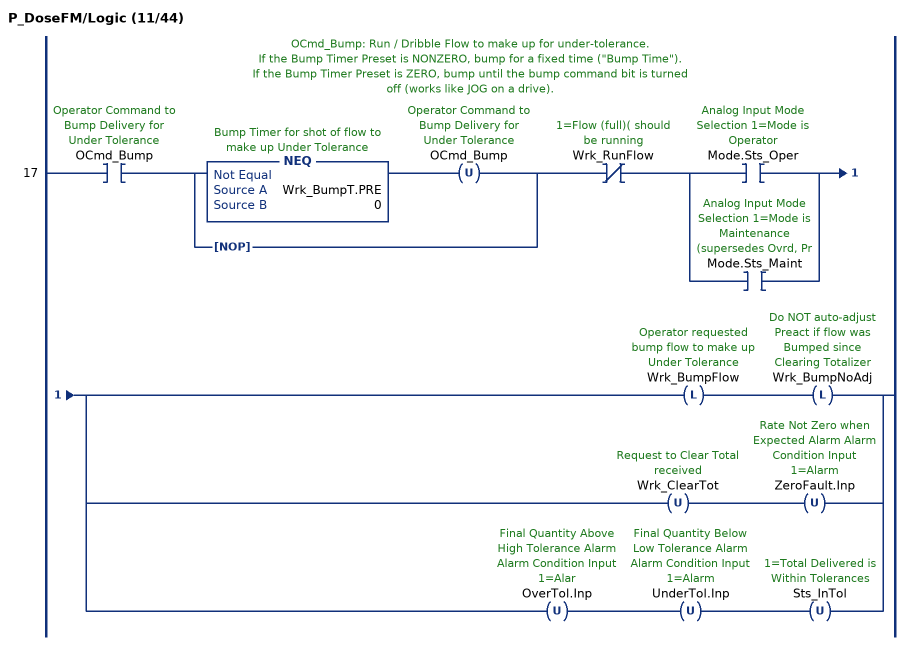
   // OCmd_Bump: Run / Dribble Flow to make up for under-tolerance.
   // If the Bump Timer Preset is NONZERO, bump for a fixed time ("Bump Time").
   // If the Bump Timer Preset is ZERO, bump until the bump command bit is turned
   // off (works like JOG on a drive).
   17: XIC(OCmd_Bump)[NEQ(Wrk_BumpT.PRE,0) OTU(OCmd_Bump) ,NOP() ]XIO(Wrk_RunFlow)[XIC(Mode.Sts_Oper) ,XIC(Mode.Sts_Maint) ][OTL(Wrk_BumpFlow) OTL(Wrk_BumpNoAdj) ,OTU(Wrk_ClearTot) OTU(ZeroFault.Inp) ,OTU(OverTol.Inp) OTU(UnderTol.Inp) OTU(Sts_InTol) ];
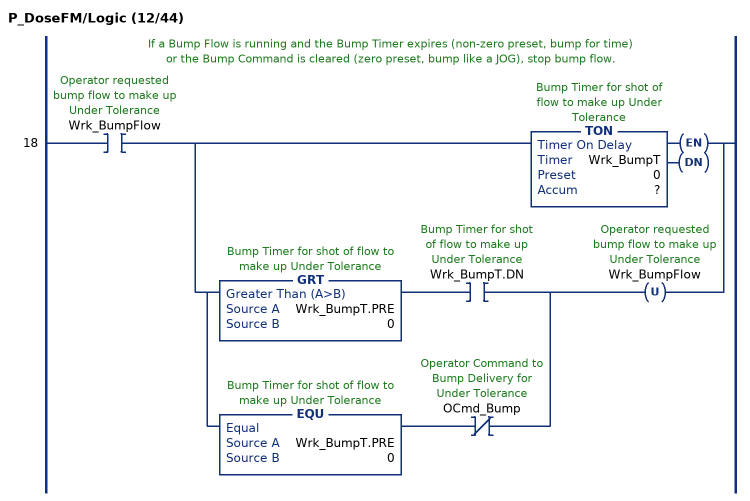
   // If a Bump Flow is running and the Bump Timer expires (non-zero preset, bump for time)
   // or the Bump Command is cleared (zero preset, bump like a JOG), stop bump flow.
   18: XIC(Wrk_BumpFlow)[TON(Wrk_BumpT,?,?) ,[GRT(Wrk_BumpT.PRE,0) XIC(Wrk_BumpT.DN) ,EQU(Wrk_BumpT.PRE,0) XIO(OCmd_Bump) ] OTU(Wrk_BumpFlow) ];
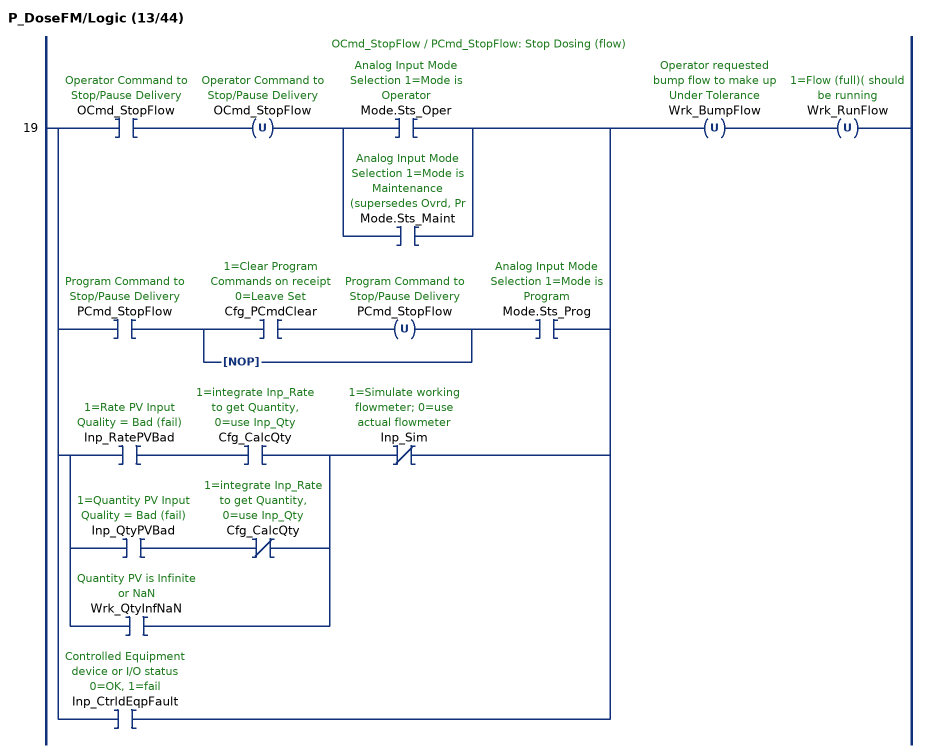
   // OCmd_StopFlow / PCmd_StopFlow: Stop Dosing (flow)
   19: [XIC(OCmd_StopFlow) OTU(OCmd_StopFlow) [XIC(Mode.Sts_Oper) ,XIC(Mode.Sts_Maint) ] ,XIC(PCmd_StopFlow) [XIC(Cfg_PCmdClear) OTU(PCmd_StopFlow) ,NOP() ] XIC(Mode.Sts_Prog) ,[XIC(Inp_RatePVBad) XIC(Cfg_CalcQty) ,XIC(Inp_QtyPVBad) XIO(Cfg_CalcQty) ,XIC(Wrk_QtyInfNaN) ] XIO(Inp_Sim) ,XIC(Inp_CtrldEqpFault) ]OTU(Wrk_BumpFlow)OTU(Wrk_RunFlow);
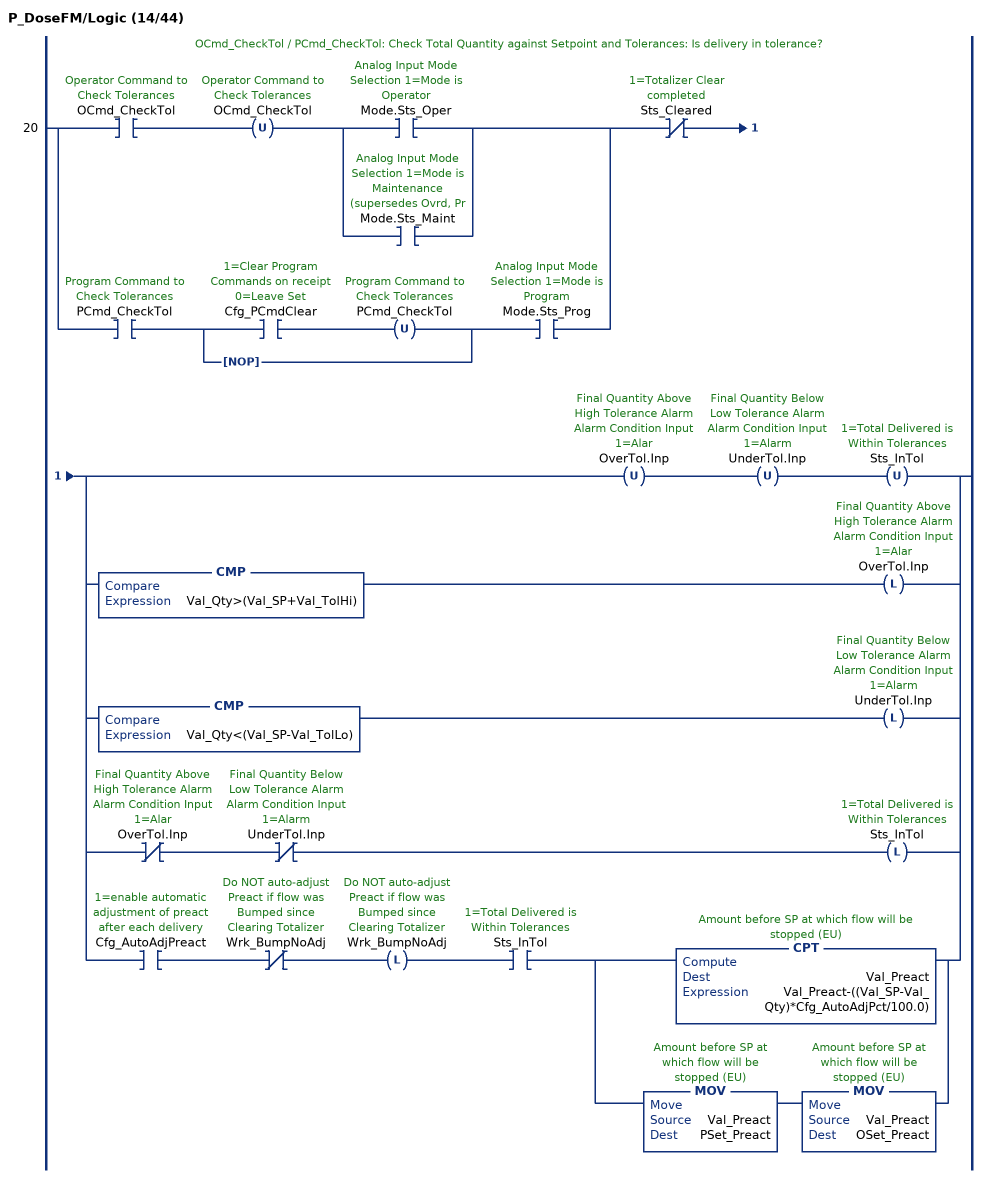
   // OCmd_CheckTol / PCmd_CheckTol: Check Total Quantity against Setpoint and Tolerances: Is delivery in tolerance?
   20: [XIC(OCmd_CheckTol) OTU(OCmd_CheckTol) [XIC(Mode.Sts_Oper) ,XIC(Mode.Sts_Maint) ] ,XIC(PCmd_CheckTol) [XIC(Cfg_PCmdClear) OTU(PCmd_CheckTol) ,NOP() ] XIC(Mode.Sts_Prog) ]XIO(Sts_Cleared)[OTU(OverTol.Inp) OTU(UnderTol.Inp) OTU(Sts_InTol) ,CMP(Val_Qty>(Val_SP+Val_TolHi)) OTL(OverTol.Inp) ,CMP(Val_Qty<(Val_SP-Val_TolLo)) OTL(UnderTol.Inp) ,XIO(OverTol.Inp) XIO(UnderTol.Inp) OTL(Sts_InTol) ,XIC(Cfg_AutoAdjPreact) XIO(Wrk_BumpNoAdj) OTL(Wrk_BumpNoAdj) XIC(Sts_InTol) [CPT(Val_Preact,Val_Preact-((Val_SP-Val_Qty)*Cfg_AutoAdjPct/100.0)) ,MOV(Val_Preact,PSet_Preact) MOV(Val_Preact,OSet_Preact) ] ];
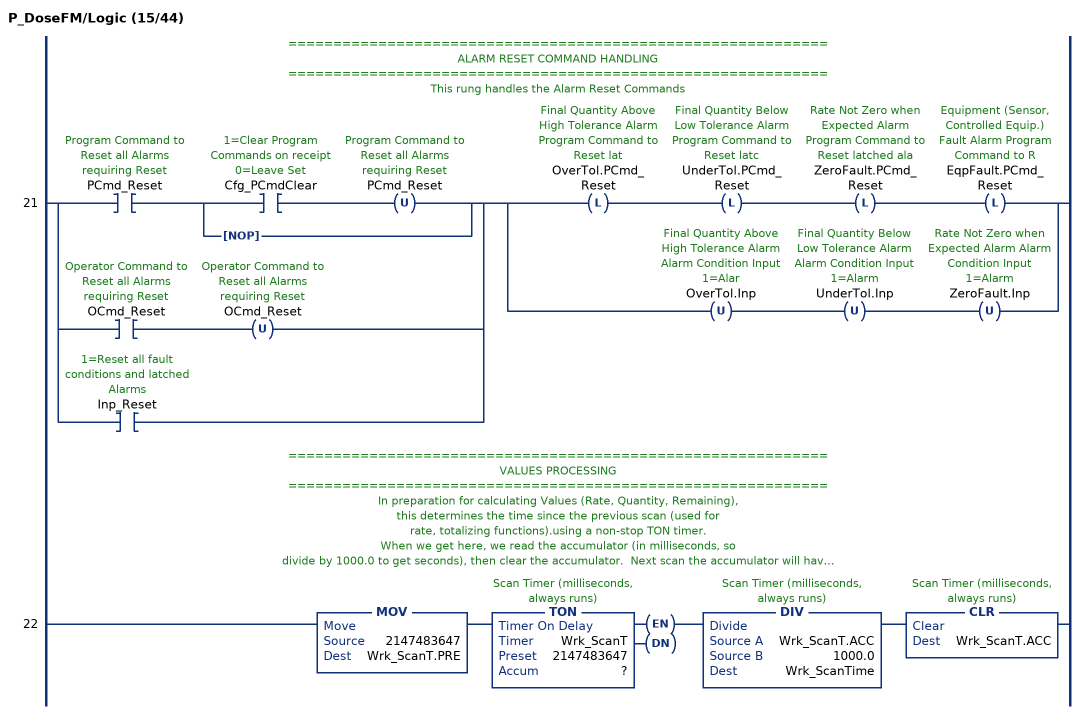
   // ============================================================
   // ALARM RESET COMMAND HANDLING
   // ============================================================
   // This rung handles the Alarm Reset Commands
   21: [XIC(PCmd_Reset) [XIC(Cfg_PCmdClear) OTU(PCmd_Reset) ,NOP() ] ,XIC(OCmd_Reset) OTU(OCmd_Reset) ,XIC(Inp_Reset) ][OTL(OverTol.PCmd_Reset) OTL(UnderTol.PCmd_Reset) OTL(ZeroFault.PCmd_Reset) OTL(EqpFault.PCmd_Reset) ,OTU(OverTol.Inp) OTU(UnderTol.Inp) OTU(ZeroFault.Inp) ];
   // ============================================================
   // VALUES PROCESSING
   // ============================================================
   // In preparation for calculating Values (Rate, Quantity, Remaining),
   // this determines the time since the previous scan (used for
   // rate, totalizing functions).using a non-stop TON timer.
   // When we get here, we read the accumulator (in milliseconds, so
   // divide by 1000.0 to get seconds), then clear the accumulator.  Next scan the accumulator will have
   // incremented up to the number of milliseconds since last scan.  (Works for scan times up to 2 million seconds.....)
   22: MOV(2147483647,Wrk_ScanT.PRE)TON(Wrk_ScanT,?,?)DIV(Wrk_ScanT.ACC,1000.0,Wrk_ScanTime)CLR(Wrk_ScanT.ACC);
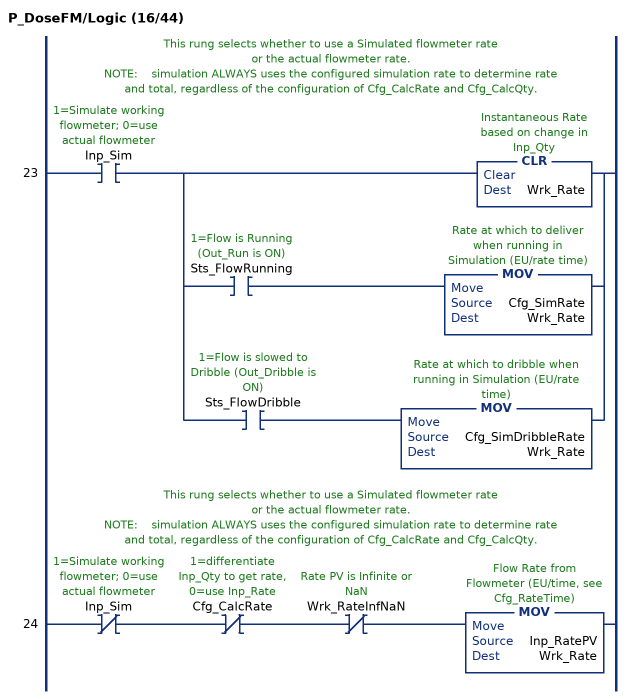
   // This rung selects whether to use a Simulated flowmeter rate
   // or the actual flowmeter rate.
   // NOTE:    simulation ALWAYS uses the configured simulation rate to determine rate
   // and total, regardless of the configuration of Cfg_CalcRate and Cfg_CalcQty.
   23: XIC(Inp_Sim)[CLR(Wrk_Rate) ,XIC(Sts_FlowRunning) MOV(Cfg_SimRate,Wrk_Rate) ,XIC(Sts_FlowDribble) MOV(Cfg_SimDribbleRate,Wrk_Rate) ];
   // This rung selects whether to use a Simulated flowmeter rate
   // or the actual flowmeter rate.
   // NOTE:    simulation ALWAYS uses the configured simulation rate to determine rate
   // and total, regardless of the configuration of Cfg_CalcRate and Cfg_CalcQty.
   24: XIO(Inp_Sim)XIO(Cfg_CalcRate)XIO(Wrk_RateInfNaN)MOV(Inp_RatePV,Wrk_Rate);
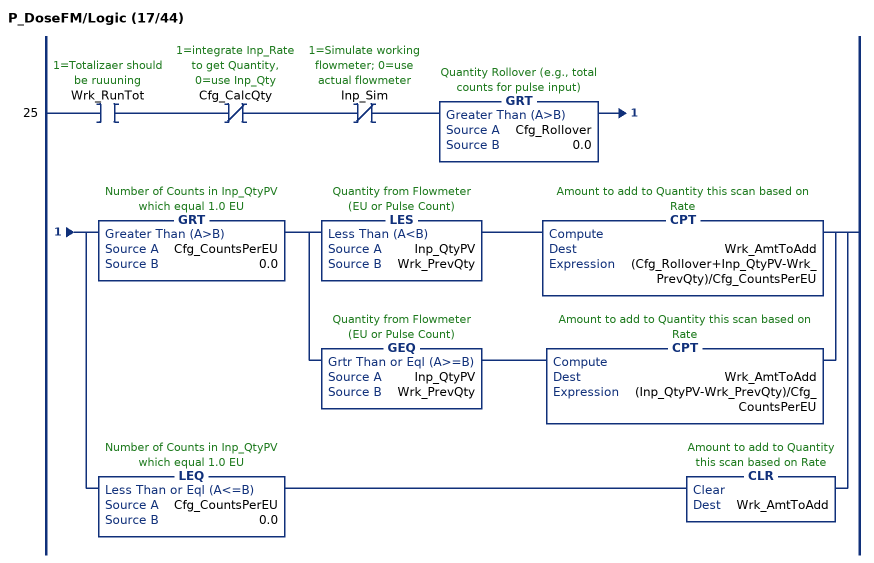
   25: XIC(Wrk_RunTot)XIO(Cfg_CalcQty)XIO(Inp_Sim)GRT(Cfg_Rollover,0.0)[GRT(Cfg_CountsPerEU,0.0) [LES(Inp_QtyPV,Wrk_PrevQty) CPT(Wrk_AmtToAdd,(Cfg_Rollover+Inp_QtyPV-Wrk_PrevQty)/Cfg_CountsPerEU) ,GEQ(Inp_QtyPV,Wrk_PrevQty) CPT(Wrk_AmtToAdd,(Inp_QtyPV-Wrk_PrevQty)/Cfg_CountsPerEU) ] ,LEQ(Cfg_CountsPerEU,0.0) CLR(Wrk_AmtToAdd) ];
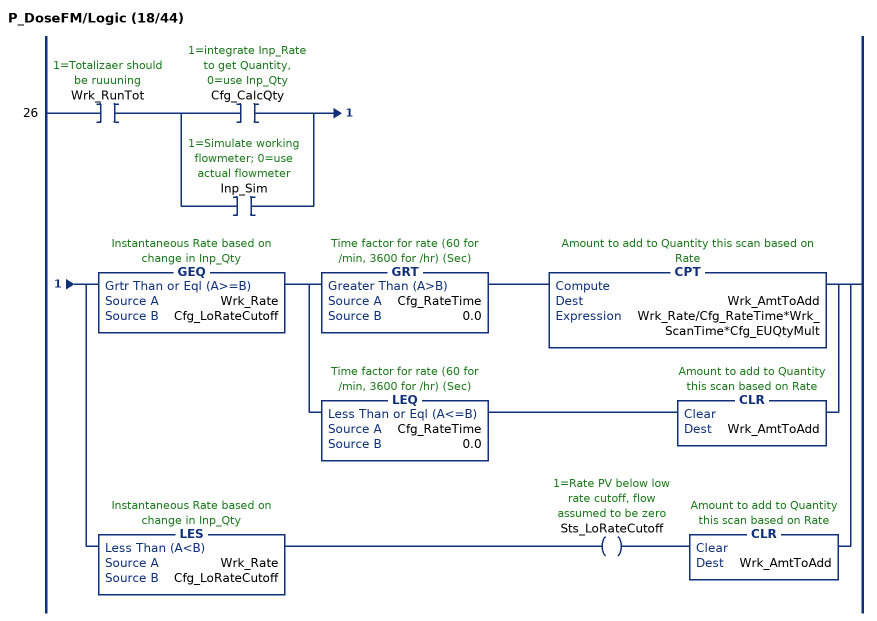
   26: XIC(Wrk_RunTot)[XIC(Cfg_CalcQty) ,XIC(Inp_Sim) ][GEQ(Wrk_Rate,Cfg_LoRateCutoff) [GRT(Cfg_RateTime,0.0) CPT(Wrk_AmtToAdd,Wrk_Rate/Cfg_RateTime*Wrk_ScanTime*Cfg_EUQtyMult) ,LEQ(Cfg_RateTime,0.0) CLR(Wrk_AmtToAdd) ] ,LES(Wrk_Rate,Cfg_LoRateCutoff) OTE(Sts_LoRateCutoff) CLR(Wrk_AmtToAdd) ];
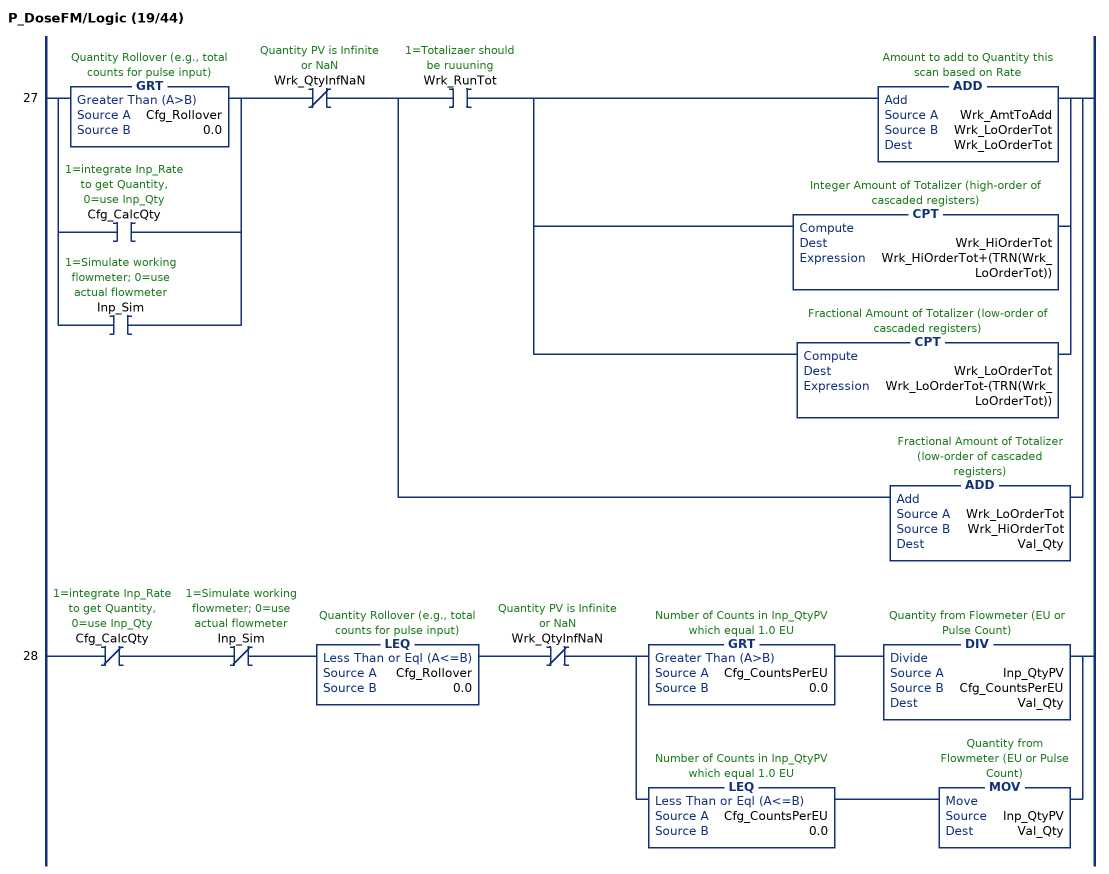
   27: [GRT(Cfg_Rollover,0.0) ,XIC(Cfg_CalcQty) ,XIC(Inp_Sim) ]XIO(Wrk_QtyInfNaN)[XIC(Wrk_RunTot) [ADD(Wrk_AmtToAdd,Wrk_LoOrderTot,Wrk_LoOrderTot) ,CPT(Wrk_HiOrderTot,Wrk_HiOrderTot+(TRN(Wrk_LoOrderTot))) ,CPT(Wrk_LoOrderTot,Wrk_LoOrderTot-(TRN(Wrk_LoOrderTot))) ] ,ADD(Wrk_LoOrderTot,Wrk_HiOrderTot,Val_Qty) ];
   28: XIO(Cfg_CalcQty)XIO(Inp_Sim)LEQ(Cfg_Rollover,0.0)XIO(Wrk_QtyInfNaN)[GRT(Cfg_CountsPerEU,0.0) DIV(Inp_QtyPV,Cfg_CountsPerEU,Val_Qty) ,LEQ(Cfg_CountsPerEU,0.0) MOV(Inp_QtyPV,Val_Qty) ];
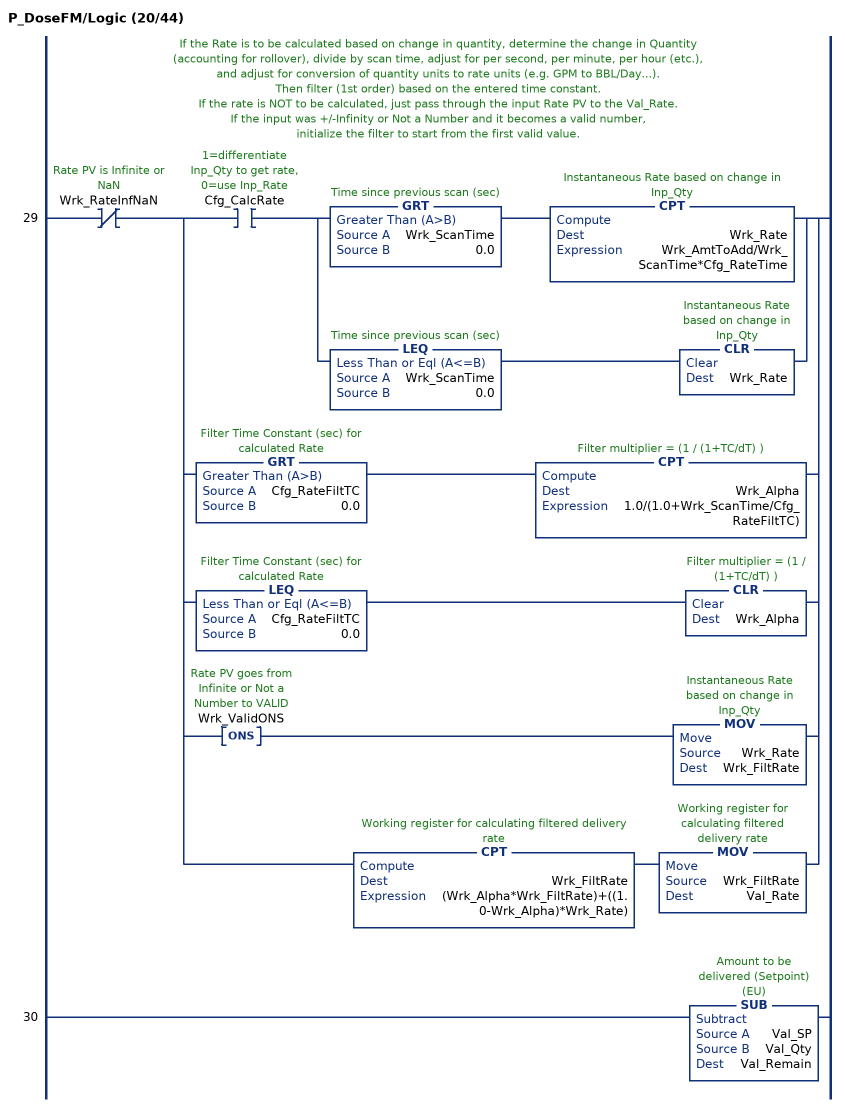
   // If the Rate is to be calculated based on change in quantity, determine the change in Quantity
   // (accounting for rollover), divide by scan time, adjust for per second, per minute, per hour (etc.),
   // and adjust for conversion of quantity units to rate units (e.g. GPM to BBL/Day...).
   // Then filter (1st order) based on the entered time constant.
   // If the rate is NOT to be calculated, just pass through the input Rate PV to the Val_Rate.
   // If the input was +/-Infinity or Not a Number and it becomes a valid number,
   // initialize the filter to start from the first valid value.
   29: XIO(Wrk_RateInfNaN)[XIC(Cfg_CalcRate) [GRT(Wrk_ScanTime,0.0) CPT(Wrk_Rate,Wrk_AmtToAdd/Wrk_ScanTime*Cfg_RateTime) ,LEQ(Wrk_ScanTime,0.0) CLR(Wrk_Rate) ] ,GRT(Cfg_RateFiltTC,0.0) CPT(Wrk_Alpha,1.0/(1.0+Wrk_ScanTime/Cfg_RateFiltTC)) ,LEQ(Cfg_RateFiltTC,0.0) CLR(Wrk_Alpha) ,ONS(Wrk_ValidONS) MOV(Wrk_Rate,Wrk_FiltRate) ,CPT(Wrk_FiltRate,(Wrk_Alpha*Wrk_FiltRate)+((1.0-Wrk_Alpha)*Wrk_Rate)) MOV(Wrk_FiltRate,Val_Rate) ];
   30: SUB(Val_SP,Val_Qty,Val_Remain);
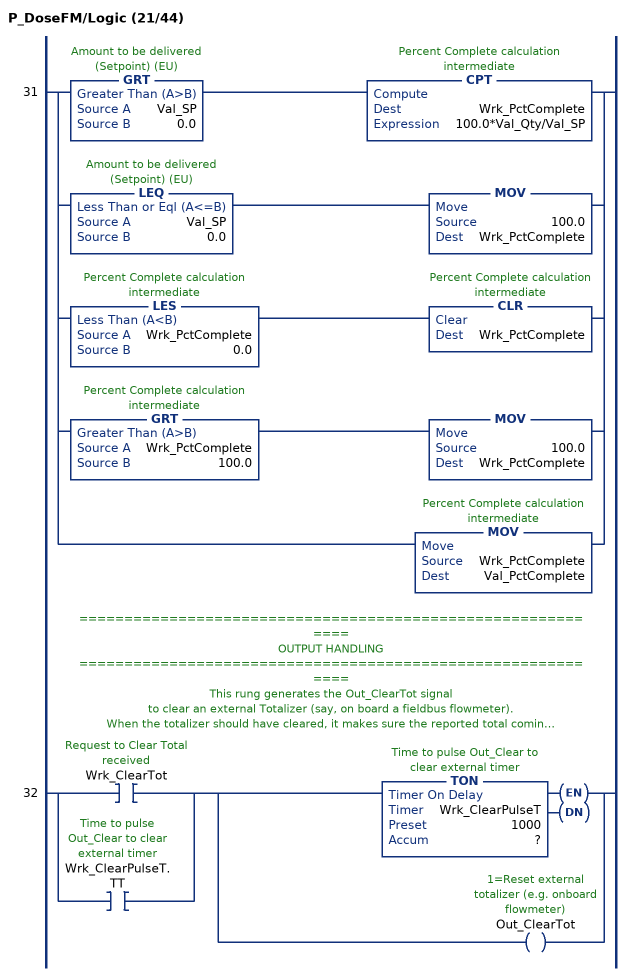
   31: [GRT(Val_SP,0.0) CPT(Wrk_PctComplete,100.0*Val_Qty/Val_SP) ,LEQ(Val_SP,0.0) MOV(100.0,Wrk_PctComplete) ,LES(Wrk_PctComplete,0.0) CLR(Wrk_PctComplete) ,GRT(Wrk_PctComplete,100.0) MOV(100.0,Wrk_PctComplete) ,MOV(Wrk_PctComplete,Val_PctComplete) ];
   // ============================================================
   // OUTPUT HANDLING
   // ============================================================
   // This rung generates the Out_ClearTot signal
   // to clear an external Totalizer (say, on board a fieldbus flowmeter).
   // When the totalizer should have cleared, it makes sure the reported total coming
   // back from the device is zero (or the internal totalizer cleared and did not count up).
   32: [XIC(Wrk_ClearTot) ,XIC(Wrk_ClearPulseT.TT) ][TON(Wrk_ClearPulseT,?,?) ,OTE(Out_ClearTot) ];
